FUNCTION_BLOCK FB_MotorControl

VAR_INPUT
	bEnable 		: BOOL;        				//FB Enable
    
    nPosition    	: LREAL;
    nVelocity    	: LREAL;
END_VAR

VAR_OUTPUT
	bDone        	: BOOL; 	//Moviment Done
    bBusy        	: BOOL;
	bPowerStatus 	: BOOL;
    bError       	: BOOL;
    nErrorID     	: UDINT;
END_VAR

VAR_IN_OUT
	AxisRef        	: AXIS_REF;	//Axis to move
END_VAR

VAR
	fbPower       	: MC_Power;         	// Habilita o motor
	MoveCommand 	: MC_MoveAbsolute; 		// Comando para movimento absoluto
	nState			: INT := 1;
	bMovDone		: BOOL := FALSE;
	bMovBusy		: BOOL := FALSE;
	bMovActive		: BOOL := FALSE;
	bMovAborted		: BOOL := FALSE;
	bMovError		: BOOL := FALSE;
	nMovErrorID		: UDINT;
END_VAR

//Powers up the axis
CASE  nState OF
	
1:
	fbPower(
    	Enable 			:= bEnable,
		Enable_Positive := bEnable,
		Enable_Negative	:= bEnable,
		Override        := 100,
    	Axis 			:= AxisRef,
    	Status 			=> bPowerStatus,
    	Error			=> bError,
    	ErrorID 		=> nErrorID
	);
	
	IF bPowerStatus THEN
		nState := 2;
	END_IF

2:
	// Verifica se o comando Start foi acionado
	IF bEnable THEN
    	MoveCommand(
			Execute 		:= TRUE,
			Axis 			:= AxisRef,
    		Position 		:= nPosition,
    		Velocity 		:= nVelocity,
    		Done 			=> bMovDone,
			Busy      		=> bMovBusy,    
    		Active     		=> bMovActive,    
    		CommandAborted	=> bMovAborted,
    		Error     		=> bMovError,     
   			ErrorID       	=> nMovErrorID
		);
	ELSE
    	MoveCommand.Execute := FALSE;
	END_IF;
	
END_CASE

END_FUNCTION_BLOCK

(* stored: Version 1.1.0.1, ProductVersion 3.1.4024.12
   POU FB_MotorControl: Id {5ab8d8f9-5e90-44d2-bb73-989aa2470e6f}, SpecialFunc None *)
